Yaskawa INFORM job: TESR8888.JBI

/JOB
//NAME TESR8888
//POS
///NPOS 12,12,12,3,0,0
///TOOL 0
///POSTYPE PULSE
///PULSE
C00000=-66856,37519,78895,-30557,64906,40783
C00001=-67664,29814,67121,-29952,67506,39742
C00002=-66312,38490,80046,-30534,64898,40987
C00003=-66205,35381,74422,-30115,66550,40552
C00004=-66856,37519,78895,-30557,64906,40783
C00005=-66037,29300,70176,-30202,66156,40726
C00006=-67455,29393,70273,-30377,65697,40331
C00007=-66037,29300,70176,-30202,66156,40726
C00008=-66241,33803,76787,-30620,64568,41109
C00009=-66037,29300,70176,-30202,66156,40726
C00010=-67131,32575,75408,-30694,64474,40808
C00011=-67599,40851,83890,-30986,63493,40924
BC00000=234833,674193,561439
BC00001=234833,674193,543158
BC00002=234833,674193,561439
BC00003=234833,674193,543556
BC00004=234833,674193,561439
BC00005=234833,674193,561439
BC00006=234833,674193,561439
BC00007=234833,674193,561439
BC00008=234833,674193,561439
BC00009=234833,674193,561439
BC00010=234833,674193,561437
BC00011=234833,674193,561437
EC00000=798145,1112941
EC00001=798145,1112941
EC00002=798145,1112941
EC00003=798145,1112941
EC00004=798145,1112941
EC00005=798145,1112941
EC00006=798145,1112941
EC00007=798145,1112941
EC00008=798145,1112941
EC00009=798145,1112941
EC00010=798144,1112940
EC00011=798144,1112940
///POSTYPE BASE
///RECTAN
///RCONF 0,0,0,0,0,0,0,0,0,0,0,0,0,0,0,0,0,0,0,0,0,0,0,0
P00006=0.222,-3.123,-1.508,0.0000,0.0000,0.0000
P00031=1.853,-0.001,-1.549,0.0000,0.0000,0.0000
P00032=1.957,0.503,-7.217,0.0000,0.0000,0.0000
//INST
///DATE 2024/03/06 15:03
///ATTR SC,RW
///GROUP1 RB1,BS1
///GROUP2 ST1
NOP
SFTOF
SSFTOF
SFTOF3D
MOVL C00000 BC00000 V=10.0  +MOVJ EC00000 VJ=0.78
SREFP 3 C00001 BC00001  +REFP EC00001
CALL JOB:SEARCH-R1-S13D
SET P031 P006
SFTON3D P031
MOVL C00002 BC00002 V=10.0  +MOVJ EC00002 VJ=0.78
SREFP 3 C00003 BC00003  +REFP EC00003
CALL JOB:SEARCH-R1-S13D
SET P031 P006
SFTOF3D
MOVL C00004 BC00004 V=11.7  +MOVJ EC00004 VJ=0.78
MOVL C00005 BC00005 V=11.7  +MOVJ EC00005 VJ=0.78
SREFP 3 C00006 BC00006  +REFP EC00006
CALL JOB:SEARCH-R1-S13D
SET P032 P006
SFTON3D P032
MOVL C00007 BC00007 V=10.0  +MOVJ EC00007 VJ=0.78
SREFP 3 C00008 BC00008  +REFP EC00008
CALL JOB:SEARCH-R1-S13D
SET P032 P006
SFTOF3D
MOVL C00009 BC00009 V=11.7  +MOVJ EC00009 VJ=0.78
PAUSE
SFTOF
SSFTOF
SFTOF3D
SFTOF
SFTON3D RB1 P032
SMOVL C00010 BC00010 V=10.0  +MOVJ EC00010
SFTOF3D
SFTON3D RB1 P031
SMOVL C00011 BC00011 V=10.0  +MOVJ EC00011
SFTOF3D
SFTOF
END
